FUNCTION_BLOCK TEST_LIM (* Test IEC 61131 LIMIT functions *)
  (* Standard: 61499-1 *)
  (* Version 0.0, 2006-09-06, JHC, Holobloc Inc *)
  (* Compiler header: package fb.rt.test; *)
  (* Compiler classdef: public class Simple extends SimpleFB *)
  (* Compiler Java Sun JDK 1.5.0 *)
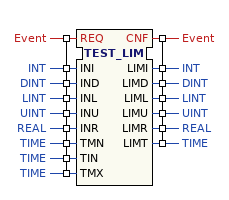
  EVENT_INPUT
    REQ WITH INI, INR, IND, INL, TIN, INU, TMN, TMX; (* Normal Execution Request *)
  END_EVENT
  EVENT_OUTPUT
    CNF WITH LIMI, LIMR, LIMD, LIML, LIMT, LIMU; (* Execution Confirmation *)
  END_EVENT
  VAR_INPUT
    INI : INT;
    IND : DINT;
    INL : LINT;
    INU : UINT;
    INR : REAL;
    TMN : TIME;
    TIN : TIME;
    TMX : TIME;
  END_VAR
  VAR_OUTPUT
    LIMI : INT; (* Output event qualifier *)
    LIMD : DINT;
    LIML : LINT;
    LIMU : UINT;
    LIMR : REAL;
    LIMT : TIME;
  END_VAR
  ALGORITHM REQ IN FBD: (* Normally executed algorithm *)
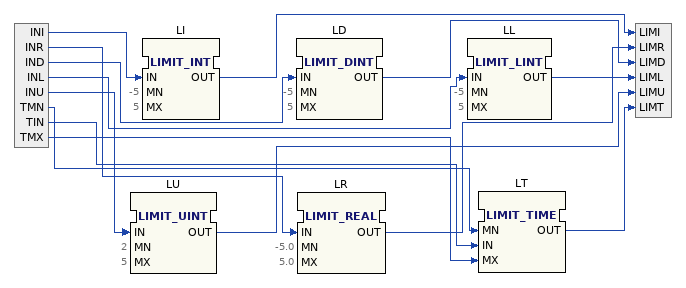
    FBS
      LI : LIMIT_INT(MN := -5, MX := 5);
      LR : LIMIT_REAL(MN := -5.0, MX := 5.0);
      LL : LIMIT_LINT(MN := -5, MX := 5);
      LT : LIMIT_TIME;
      LU : LIMIT_UINT(MN := 2, MX := 5);
      LD : LIMIT_DINT(MN := -5, MX := 5);
    END_FBS
    DATA_CONNECTIONS
      INI TO LI.IN;
      LI.OUT TO LIMI;
      INR TO LR.IN;
      LR.OUT TO LIMR;
      IND TO LD.IN;
      LD.OUT TO LIMD;
      INL TO LL.IN;
      LL.OUT TO LIML;
      INU TO LU.IN;
      LU.OUT TO LIMU;
      LT.OUT TO LIMT;
      TMN TO LT.MN;
      TIN TO LT.IN;
      TMX TO LT.MX;
    END_CONNECTIONS
  END_ALGORITHM
END_FUNCTION_BLOCK
